TYPE ST_StatusDI :
STRUCT
	RawValue					: BOOL := FALSE;
	P_Value						: BOOL := FALSE;
END_STRUCT
END_TYPE

(* stored: Version 1.1.0.1, ProductVersion 3.1.4026.18
   DUT ST_StatusDI: Id {113e4c33-ed73-49d1-a248-1c9a38f676c0} *)
